// TIA Portal V16 export
// export: Created 2022-11-17T11:55:03.1520039Z, ExportSetting WithDefaults, DisplayName Totally Integrated Automation Portal, DisplayVersion V16 Update 6, DisplayName TIA Portal Version Control Interface, DisplayVersion V16 Update 2, DisplayName TIA Portal Openness, DisplayVersion V16 Update 6, DisplayName SINAMICS Startdrive Advanced, DisplayVersion V16 Update 5, DisplayName SINAMICS Startdrive G130, G150, S120, S150, SINAMICS MV, S210, DisplayVersion V16 Update 5, DisplayName SINAMICS Startdrive G110M, G120, G120C, G120D, G120P, G115D, DisplayVersion V16 Update 5, DisplayName STEP 7 Professional, DisplayVersion V16 Update 6, DisplayName STEP 7 Safety, DisplayVersion V16, DisplayName WinCC Advanced, DisplayVersion V16 Update 6
FUNCTION "FC04_TechnoplatAlarm" : Void   // FC4, LAD
TITLE = Alarm for the machine
{ S7_Optimized_Access := 'FALSE' }
AUTHOR : Robopac
VERSION : 0.0
// stored: AutoNumber false, IsIECCheckEnabled false, SetENOAutomatically false, UDAEnableTagReadback false
BEGIN

REGION Network 1: Alarm 1: Pressure switch (Technoplat)
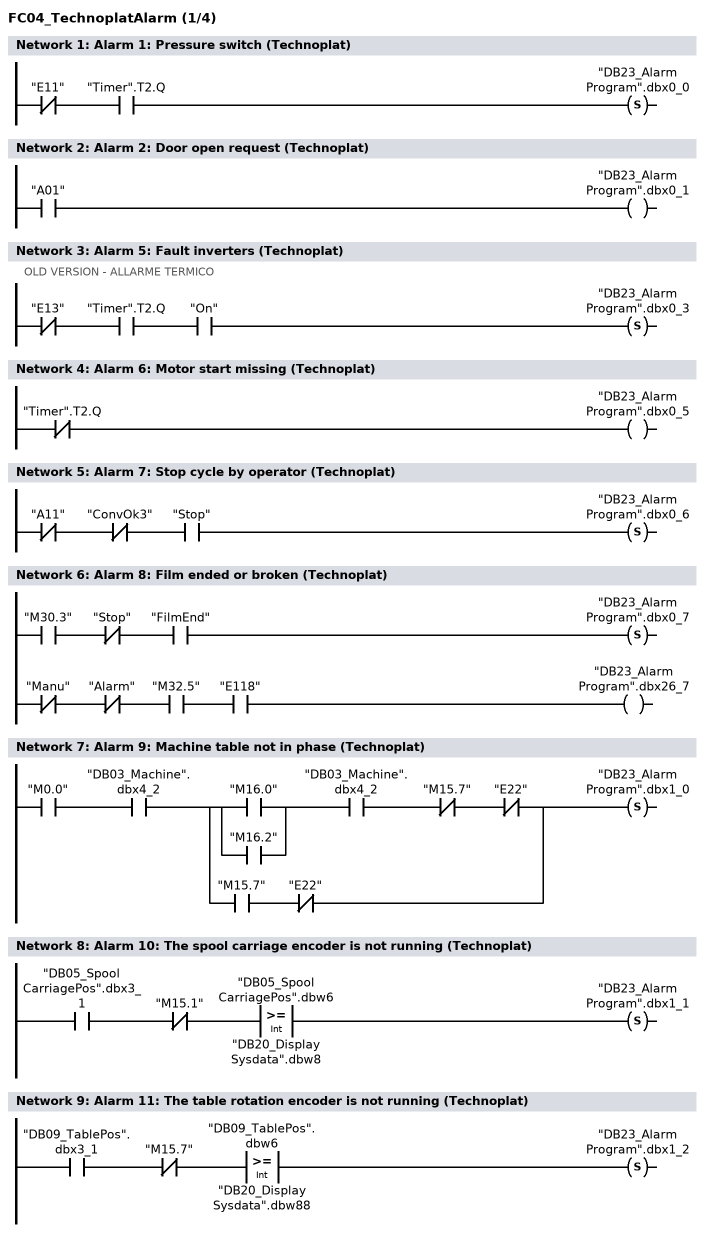
   RUNG wire#powerrail
      I_Contact( "E11" )
      Contact( "Timer".T2.Q )
      S_Coil( "DB23_AlarmProgram".dbx0_0 )
   END_RUNG
   // the same network as SCL:
   IF NOT "E11" AND "Timer".T2.Q THEN "DB23_AlarmProgram".dbx0_0 := TRUE; END_IF;
END_REGION

REGION Network 2: Alarm 2: Door open request (Technoplat)
   RUNG wire#powerrail
      Contact( "A01" )
      Coil( "DB23_AlarmProgram".dbx0_1 )
   END_RUNG
   // the same network as SCL:
   "DB23_AlarmProgram".dbx0_1 := "A01";
END_REGION

REGION Network 3: Alarm 5: Fault inverters (Technoplat)
   // OLD VERSION - ALLARME TERMICO
   RUNG wire#powerrail
      I_Contact( "E13" )
      Contact( "Timer".T2.Q )
      Contact( "On" )
      S_Coil( "DB23_AlarmProgram".dbx0_3 )
   END_RUNG
   // the same network as SCL:
   IF NOT "E13" AND "Timer".T2.Q AND "On" THEN "DB23_AlarmProgram".dbx0_3 := TRUE; END_IF;
END_REGION

REGION Network 4: Alarm 6: Motor start missing (Technoplat)
   RUNG wire#powerrail
      I_Contact( "Timer".T2.Q )
      Coil( "DB23_AlarmProgram".dbx0_5 )
   END_RUNG
   // the same network as SCL:
   "DB23_AlarmProgram".dbx0_5 := NOT "Timer".T2.Q;
END_REGION

REGION Network 5: Alarm 7: Stop cycle by operator (Technoplat)
   RUNG wire#powerrail
      I_Contact( "A11" )
      I_Contact( "ConvOk3" )
      Contact( "Stop" )
      S_Coil( "DB23_AlarmProgram".dbx0_6 )
   END_RUNG
   // the same network as SCL:
   IF NOT "A11" AND NOT "ConvOk3" AND "Stop" THEN "DB23_AlarmProgram".dbx0_6 := TRUE; END_IF;
END_REGION

REGION Network 6: Alarm 8: Film ended or broken (Technoplat)
   RUNG wire#powerrail
      Contact( "M30.3" )
      I_Contact( "Stop" )
      Contact( "FilmEnd" )
      S_Coil( "DB23_AlarmProgram".dbx0_7 )
   END_RUNG
   RUNG wire#powerrail
      I_Contact( "Manu" )
      I_Contact( "Alarm" )
      Contact( "M32.5" )
      Contact( "E118" )
      Coil( "DB23_AlarmProgram".dbx26_7 )
   END_RUNG
   // the same network as SCL:
   IF "M30.3" AND NOT "Stop" AND "FilmEnd" THEN "DB23_AlarmProgram".dbx0_7 := TRUE; END_IF;
   "DB23_AlarmProgram".dbx26_7 := NOT "Manu" AND NOT "Alarm" AND "M32.5" AND "E118";
END_REGION

REGION Network 7: Alarm 9: Machine table not in phase (Technoplat)
   RUNG wire#powerrail
      Contact( "M0.0" )
      Contact( "DB03_Machine".dbx4_2 )
      wire#w1
      Contact( "M16.0" )
      wire#w2
      Contact( "DB03_Machine".dbx4_2 )
      I_Contact( "M15.7" )
      I_Contact( "E22" )
      wire#w3
      S_Coil( "DB23_AlarmProgram".dbx1_0 )
   END_RUNG
   RUNG wire#w1
      Contact( "M16.2" )
   END_RUNG wire#w2
   RUNG wire#w1
      Contact( "M15.7" )
      I_Contact( "E22" )
   END_RUNG wire#w3
   // the same network as SCL:
   IF "M0.0" AND "DB03_Machine".dbx4_2 AND ((("M16.0" OR "M16.2") AND "DB03_Machine".dbx4_2 AND NOT "M15.7" AND NOT "E22") OR ("M15.7" AND NOT "E22")) THEN
       "DB23_AlarmProgram".dbx1_0 := TRUE;
   END_IF;
END_REGION

REGION Network 8: Alarm 10: The spool carriage encoder is not running (Technoplat)
   RUNG wire#powerrail
      Contact( "DB05_SpoolCarriagePos".dbx3_1 )
      I_Contact( "M15.1" )
      { S7_Templates := "SrcType := Int" } GE_Contact(in1 := "DB05_SpoolCarriagePos".dbw6, in2 := "DB20_DisplaySysdata".dbw8)
      S_Coil( "DB23_AlarmProgram".dbx1_1 )
   END_RUNG
   // the same network as SCL:
   IF "DB05_SpoolCarriagePos".dbx3_1 AND NOT "M15.1" AND ("DB05_SpoolCarriagePos".dbw6 >= "DB20_DisplaySysdata".dbw8) THEN
       "DB23_AlarmProgram".dbx1_1 := TRUE;
   END_IF;
END_REGION

REGION Network 9: Alarm 11: The table rotation encoder is not running (Technoplat)
   RUNG wire#powerrail
      Contact( "DB09_TablePos".dbx3_1 )
      I_Contact( "M15.7" )
      { S7_Templates := "SrcType := Int" } GE_Contact(in1 := "DB09_TablePos".dbw6, in2 := "DB20_DisplaySysdata".dbw88)
      S_Coil( "DB23_AlarmProgram".dbx1_2 )
   END_RUNG
   // the same network as SCL:
   IF "DB09_TablePos".dbx3_1 AND NOT "M15.7" AND ("DB09_TablePos".dbw6 >= "DB20_DisplaySysdata".dbw88) THEN
       "DB23_AlarmProgram".dbx1_2 := TRUE;
   END_IF;
END_REGION

REGION Network 10: Alarm 12: Overspeed for arm rotation (Technoplat)
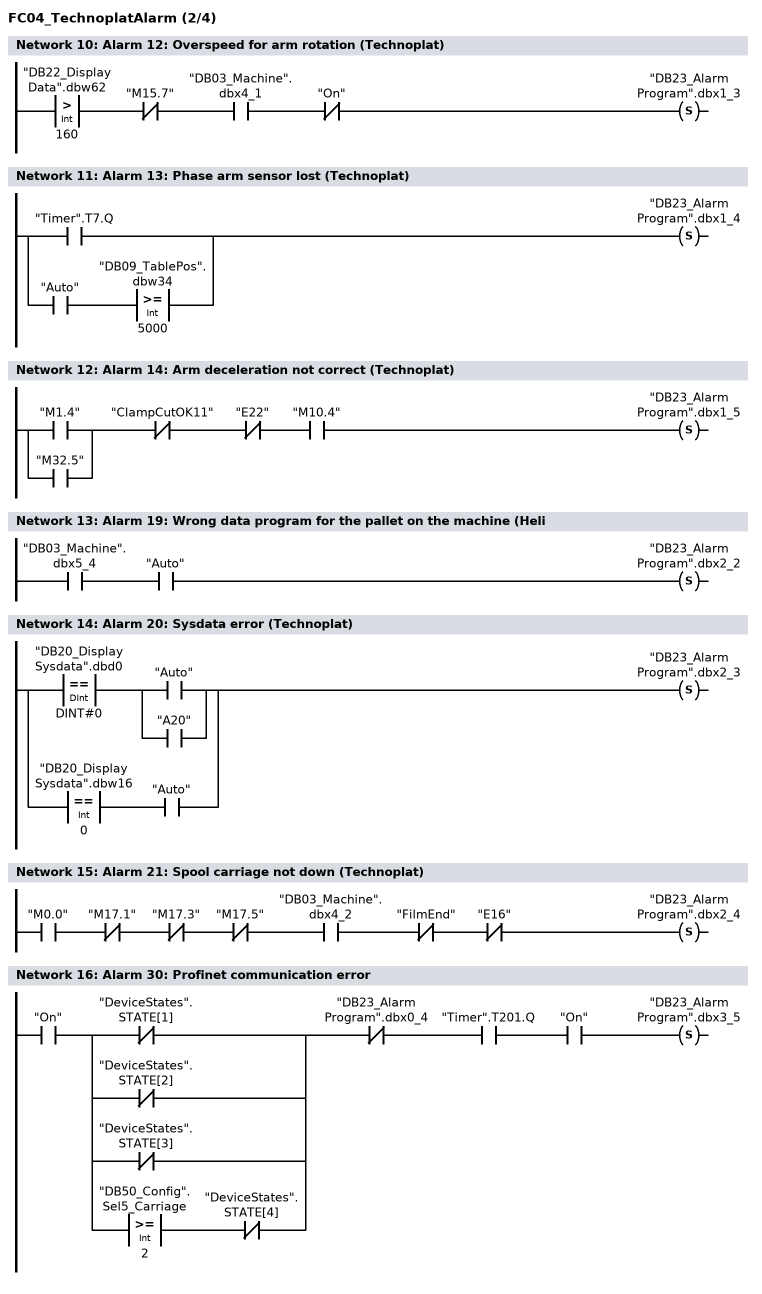
   RUNG wire#powerrail
      { S7_Templates := "SrcType := Int" } GT_Contact(in1 := "DB22_DisplayData".dbw62, in2 := 160)
      I_Contact( "M15.7" )
      Contact( "DB03_Machine".dbx4_1 )
      I_Contact( "On" )
      S_Coil( "DB23_AlarmProgram".dbx1_3 )
   END_RUNG
   // the same network as SCL:
   IF ("DB22_DisplayData".dbw62 > 160) AND NOT "M15.7" AND "DB03_Machine".dbx4_1 AND NOT "On" THEN
       "DB23_AlarmProgram".dbx1_3 := TRUE;
   END_IF;
END_REGION

REGION Network 11: Alarm 13: Phase arm sensor lost (Technoplat)
   RUNG wire#powerrail
      Contact( "Timer".T7.Q )
      wire#w1
      S_Coil( "DB23_AlarmProgram".dbx1_4 )
   END_RUNG
   RUNG wire#powerrail
      Contact( "Auto" )
      { S7_Templates := "SrcType := Int" } GE_Contact(in1 := "DB09_TablePos".dbw34, in2 := 5000)
   END_RUNG wire#w1
   // the same network as SCL:
   IF "Timer".T7.Q OR ("Auto" AND ("DB09_TablePos".dbw34 >= 5000)) THEN
       "DB23_AlarmProgram".dbx1_4 := TRUE;
   END_IF;
END_REGION

REGION Network 12: Alarm 14: Arm deceleration not correct (Technoplat)
   RUNG wire#powerrail
      Contact( "M1.4" )
      wire#w1
      I_Contact( "ClampCutOK11" )
      I_Contact( "E22" )
      Contact( "M10.4" )
      S_Coil( "DB23_AlarmProgram".dbx1_5 )
   END_RUNG
   RUNG wire#powerrail
      Contact( "M32.5" )
   END_RUNG wire#w1
   // the same network as SCL:
   IF ("M1.4" OR "M32.5") AND NOT "ClampCutOK11" AND NOT "E22" AND "M10.4" THEN
       "DB23_AlarmProgram".dbx1_5 := TRUE;
   END_IF;
END_REGION

REGION Network 13: Alarm 19: Wrong data program for the pallet on the machine (Heli
   RUNG wire#powerrail
      Contact( "DB03_Machine".dbx5_4 )
      Contact( "Auto" )
      S_Coil( "DB23_AlarmProgram".dbx2_2 )
   END_RUNG
   // the same network as SCL:
   IF "DB03_Machine".dbx5_4 AND "Auto" THEN "DB23_AlarmProgram".dbx2_2 := TRUE; END_IF;
END_REGION

REGION Network 14: Alarm 20: Sysdata error (Technoplat)
   RUNG wire#powerrail
      { S7_Templates := "SrcType := DInt" } EQ_Contact(in1 := "DB20_DisplaySysdata".dbd0, in2 := DINT#0)
      wire#w1
      Contact( "Auto" )
      wire#w2
      S_Coil( "DB23_AlarmProgram".dbx2_3 )
   END_RUNG
   RUNG wire#w1
      Contact( "A20" )
   END_RUNG wire#w2
   RUNG wire#powerrail
      { S7_Templates := "SrcType := Int" } EQ_Contact(in1 := "DB20_DisplaySysdata".dbw16, in2 := 0)
      Contact( "Auto" )
   END_RUNG wire#w2
   // the same network as SCL:
   IF (("DB20_DisplaySysdata".dbd0 = DINT#0) AND ("Auto" OR "A20")) OR (("DB20_DisplaySysdata".dbw16 = 0) AND "Auto") THEN
       "DB23_AlarmProgram".dbx2_3 := TRUE;
   END_IF;
END_REGION

REGION Network 15: Alarm 21: Spool carriage not down (Technoplat)
   RUNG wire#powerrail
      Contact( "M0.0" )
      I_Contact( "M17.1" )
      I_Contact( "M17.3" )
      I_Contact( "M17.5" )
      Contact( "DB03_Machine".dbx4_2 )
      I_Contact( "FilmEnd" )
      I_Contact( "E16" )
      S_Coil( "DB23_AlarmProgram".dbx2_4 )
   END_RUNG
   // the same network as SCL:
   IF "M0.0" AND NOT "M17.1" AND NOT "M17.3" AND NOT "M17.5" AND "DB03_Machine".dbx4_2 AND NOT "FilmEnd" AND NOT "E16" THEN
       "DB23_AlarmProgram".dbx2_4 := TRUE;
   END_IF;
END_REGION

REGION Network 16: Alarm 30: Profinet communication error
   RUNG wire#powerrail
      Contact( "On" )
      wire#w1
      I_Contact( "DeviceStates".STATE[1] )
      wire#w2
      I_Contact( "DB23_AlarmProgram".dbx0_4 )
      Contact( "Timer".T201.Q )
      Contact( "On" )
      S_Coil( "DB23_AlarmProgram".dbx3_5 )
   END_RUNG
   RUNG wire#w1
      I_Contact( "DeviceStates".STATE[2] )
   END_RUNG wire#w2
   RUNG wire#w1
      I_Contact( "DeviceStates".STATE[3] )
   END_RUNG wire#w2
   RUNG wire#w1
      { S7_Templates := "SrcType := Int" } GE_Contact(in1 := "DB50_Config".Sel5_Carriage, in2 := 2)
      I_Contact( "DeviceStates".STATE[4] )
   END_RUNG wire#w2
   // the same network as SCL:
   IF "On" AND (NOT "DeviceStates".STATE[1] OR NOT "DeviceStates".STATE[2] OR NOT "DeviceStates".STATE[3] OR (("DB50_Config".Sel5_Carriage >= 2) AND NOT "DeviceStates".STATE[4])) AND NOT "DB23_AlarmProgram".dbx0_4 AND "Timer".T201.Q AND "On" THEN
       "DB23_AlarmProgram".dbx3_5 := TRUE;
   END_IF;
END_REGION

REGION Network 17: Alarm 31: Modbus communication error
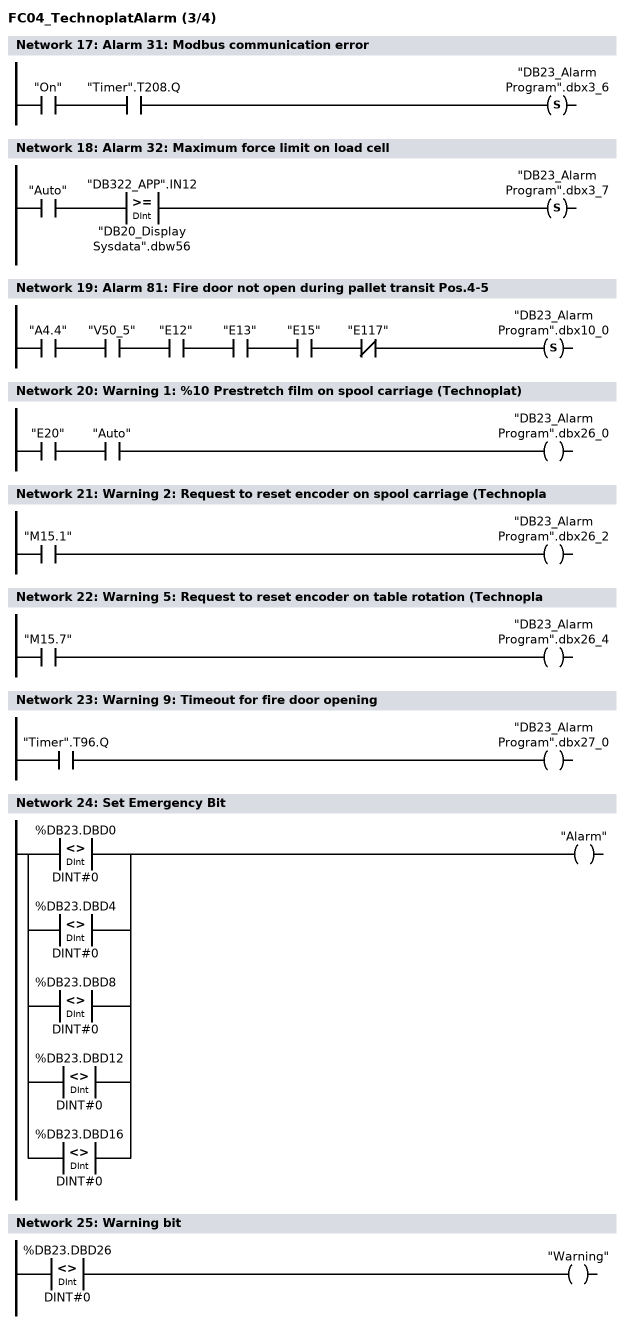
   RUNG wire#powerrail
      Contact( "On" )
      Contact( "Timer".T208.Q )
      S_Coil( "DB23_AlarmProgram".dbx3_6 )
   END_RUNG
   // the same network as SCL:
   IF "On" AND "Timer".T208.Q THEN "DB23_AlarmProgram".dbx3_6 := TRUE; END_IF;
END_REGION

REGION Network 18: Alarm 32: Maximum force limit on load cell
   RUNG wire#powerrail
      Contact( "Auto" )
      { S7_Templates := "SrcType := DInt" } GE_Contact(in1 := "DB322_APP".IN12, in2 := "DB20_DisplaySysdata".dbw56)
      S_Coil( "DB23_AlarmProgram".dbx3_7 )
   END_RUNG
   // the same network as SCL:
   IF "Auto" AND ("DB322_APP".IN12 >= "DB20_DisplaySysdata".dbw56) THEN
       "DB23_AlarmProgram".dbx3_7 := TRUE;
   END_IF;
END_REGION

REGION Network 19: Alarm 81: Fire door not open during pallet transit Pos.4-5
   RUNG wire#powerrail
      Contact( "A4.4" )
      Contact( "V50_5" )
      Contact( "E12" )
      Contact( "E13" )
      Contact( "E15" )
      I_Contact( "E117" )
      S_Coil( "DB23_AlarmProgram".dbx10_0 )
   END_RUNG
   // the same network as SCL:
   IF "A4.4" AND "V50_5" AND "E12" AND "E13" AND "E15" AND NOT "E117" THEN
       "DB23_AlarmProgram".dbx10_0 := TRUE;
   END_IF;
END_REGION

REGION Network 20: Warning 1: %10 Prestretch film on spool carriage (Technoplat)
   RUNG wire#powerrail
      Contact( "E20" )
      Contact( "Auto" )
      Coil( "DB23_AlarmProgram".dbx26_0 )
   END_RUNG
   // the same network as SCL:
   "DB23_AlarmProgram".dbx26_0 := "E20" AND "Auto";
END_REGION

REGION Network 21: Warning 2: Request to reset encoder on spool carriage (Technopla
   RUNG wire#powerrail
      Contact( "M15.1" )
      Coil( "DB23_AlarmProgram".dbx26_2 )
   END_RUNG
   // the same network as SCL:
   "DB23_AlarmProgram".dbx26_2 := "M15.1";
END_REGION

REGION Network 22: Warning 5: Request to reset encoder on table rotation (Technopla
   RUNG wire#powerrail
      Contact( "M15.7" )
      Coil( "DB23_AlarmProgram".dbx26_4 )
   END_RUNG
   // the same network as SCL:
   "DB23_AlarmProgram".dbx26_4 := "M15.7";
END_REGION

REGION Network 23: Warning 9: Timeout for fire door opening
   RUNG wire#powerrail
      Contact( "Timer".T96.Q )
      Coil( "DB23_AlarmProgram".dbx27_0 )
   END_RUNG
   // the same network as SCL:
   "DB23_AlarmProgram".dbx27_0 := "Timer".T96.Q;
END_REGION

REGION Network 24: Set Emergency Bit
   RUNG wire#powerrail
      { S7_Templates := "SrcType := DInt" } NE_Contact(in1 := %DB23.DBD0, in2 := DINT#0)
      wire#w1
      Coil( "Alarm" )
   END_RUNG
   RUNG wire#powerrail
      { S7_Templates := "SrcType := DInt" } NE_Contact(in1 := %DB23.DBD4, in2 := DINT#0)
   END_RUNG wire#w1
   RUNG wire#powerrail
      { S7_Templates := "SrcType := DInt" } NE_Contact(in1 := %DB23.DBD8, in2 := DINT#0)
   END_RUNG wire#w1
   RUNG wire#powerrail
      { S7_Templates := "SrcType := DInt" } NE_Contact(in1 := %DB23.DBD12, in2 := DINT#0)
   END_RUNG wire#w1
   RUNG wire#powerrail
      { S7_Templates := "SrcType := DInt" } NE_Contact(in1 := %DB23.DBD16, in2 := DINT#0)
   END_RUNG wire#w1
   // the same network as SCL:
   "Alarm" := (%DB23.DBD0 <> DINT#0) OR (%DB23.DBD4 <> DINT#0) OR (%DB23.DBD8 <> DINT#0) OR (%DB23.DBD12 <> DINT#0) OR (%DB23.DBD16 <> DINT#0);
END_REGION

REGION Network 25: Warning bit
   RUNG wire#powerrail
      { S7_Templates := "SrcType := DInt" } NE_Contact(in1 := %DB23.DBD26, in2 := DINT#0)
      Coil( "Warning" )
   END_RUNG
   // the same network as SCL:
   "Warning" := %DB23.DBD26 <> DINT#0;
END_REGION

REGION Network 26: First cycle
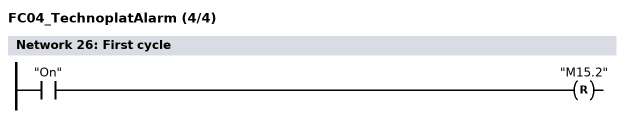
   RUNG wire#powerrail
      Contact( "On" )
      R_Coil( "M15.2" )
   END_RUNG
   // the same network as SCL:
   IF "On" THEN "M15.2" := FALSE; END_IF;
END_REGION
END_FUNCTION
